% RSLogix 500 project Project 2.RSS, saved by version 8.30.00.16 %
PROJECT "UNTITLED"    % processor: Bul.1763 MicroLogix 1100 Series B %

PROGRAM FILES
  LAD 2 "MAIN"  3 rungs
  LAD 3 "DIGITAL IO"  8 rungs
  LAD 4 "CONTROLS"  5 rungs

DATA FILES
  O0 OUTPUT  4 elements
  I1 INPUT  6 elements
  S2 STATUS  66 elements
  B3 BINARY  1 elements
  T4 TIMER  1 elements
  C5 COUNTER  1 elements
  R6 CONTROL  1 elements
  N7 INTEGER  1 elements
  F8 FLOAT  1 elements

LADDER 2 "MAIN"
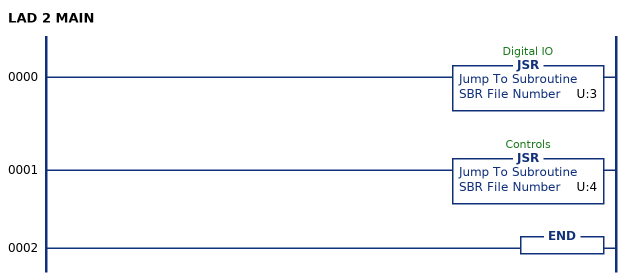
% Rung: 0 %
SOR JSR U:3 EOR
%   U:3  "Digital IO" %
% Rung: 1 %
SOR JSR U:4 EOR
%   U:4  "Controls" %
% Rung: 2 %
SOR END EOR

LADDER 3 "DIGITAL IO"
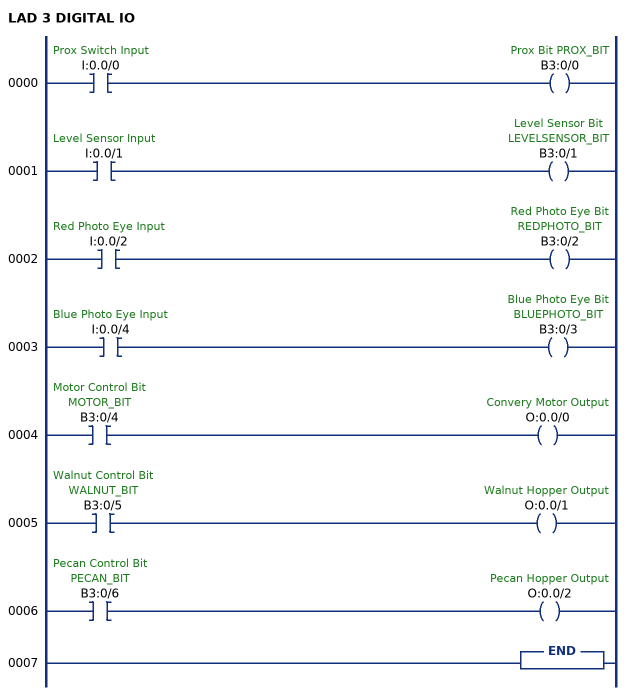
% Rung: 0 %
SOR XIC I:0.0/0 OTE B3:0/0 EOR
%   I:0.0/0  "Prox Switch Input" %
%   B3:0/0  PROX_BIT  "Prox Bit" %
% Rung: 1 %
SOR XIC I:0.0/1 OTE B3:0/1 EOR
%   I:0.0/1  "Level Sensor Input" %
%   B3:0/1  LEVELSENSOR_BIT  "Level Sensor Bit" %
% Rung: 2 %
SOR XIC I:0.0/2 OTE B3:0/2 EOR
%   I:0.0/2  "Red Photo Eye Input" %
%   B3:0/2  REDPHOTO_BIT  "Red Photo Eye Bit" %
% Rung: 3 %
SOR XIC I:0.0/4 OTE B3:0/3 EOR
%   I:0.0/4  "Blue Photo Eye Input" %
%   B3:0/3  BLUEPHOTO_BIT  "Blue Photo Eye Bit" %
% Rung: 4 %
SOR XIC B3:0/4 OTE O:0.0/0 EOR
%   B3:0/4  MOTOR_BIT  "Motor Control Bit" %
%   O:0.0/0  "Convery Motor Output" %
% Rung: 5 %
SOR XIC B3:0/5 OTE O:0.0/1 EOR
%   B3:0/5  WALNUT_BIT  "Walnut Control Bit" %
%   O:0.0/1  "Walnut Hopper Output" %
% Rung: 6 %
SOR XIC B3:0/6 OTE O:0.0/2 EOR
%   B3:0/6  PECAN_BIT  "Pecan Control Bit" %
%   O:0.0/2  "Pecan Hopper Output" %
% Rung: 7 %
SOR END EOR

LADDER 4 "CONTROLS"
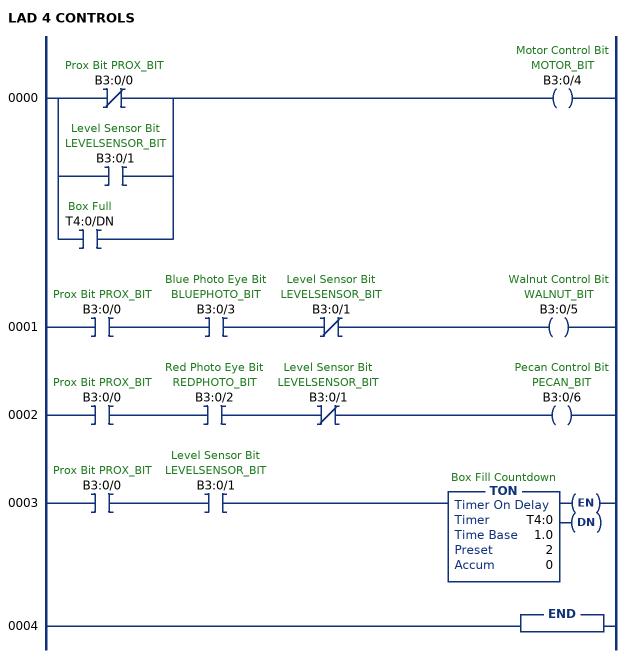
% Rung: 0 %
SOR BST XIO B3:0/0 NXB XIC B3:0/1 NXB XIC T4:0/DN BND OTE B3:0/4 EOR
%   B3:0/0  PROX_BIT  "Prox Bit" %
%   B3:0/1  LEVELSENSOR_BIT  "Level Sensor Bit" %
%   T4:0/DN  "Box Full" %
%   B3:0/4  MOTOR_BIT  "Motor Control Bit" %
% Rung: 1 %
SOR XIC B3:0/0 XIC B3:0/3 XIO B3:0/1 OTE B3:0/5 EOR
%   B3:0/0  PROX_BIT  "Prox Bit" %
%   B3:0/3  BLUEPHOTO_BIT  "Blue Photo Eye Bit" %
%   B3:0/1  LEVELSENSOR_BIT  "Level Sensor Bit" %
%   B3:0/5  WALNUT_BIT  "Walnut Control Bit" %
% Rung: 2 %
SOR XIC B3:0/0 XIC B3:0/2 XIO B3:0/1 OTE B3:0/6 EOR
%   B3:0/0  PROX_BIT  "Prox Bit" %
%   B3:0/2  REDPHOTO_BIT  "Red Photo Eye Bit" %
%   B3:0/1  LEVELSENSOR_BIT  "Level Sensor Bit" %
%   B3:0/6  PECAN_BIT  "Pecan Control Bit" %
% Rung: 3 %
SOR XIC B3:0/0 XIC B3:0/1 TON T4:0 1.0 2 0 EOR
%   B3:0/0  PROX_BIT  "Prox Bit" %
%   B3:0/1  LEVELSENSOR_BIT  "Level Sensor Bit" %
%   T4:0  "Box Fill Countdown" %
% Rung: 4 %
SOR END EOR

OTHER DOCUMENTED ADDRESSES
  B3:0/7  "Fire Once"
  B3:0/8  "Fire Once"
  B3:0/9  "Walnut Trigger Bit"
  B3:0/10  "Pecan Trigger Bit"
  B3:0/11  "Fire Once"
  N7:0  "Cycle 0 - Bring the Box 1 - Fill the Box 2 - Take the Box"
  U:5  "Cycle"

DATA TABLE (non-zero values as saved)
DATA T4
% .PRE .ACC %
% T4:0 % 2 0
